// TIA Portal V17 export
// export: Created 2024-08-20T13:26:05.2375975Z, ExportSetting WithDefaults, DisplayName Totally Integrated Automation Portal, DisplayVersion V17 Update 4, DisplayName TIA Portal Openness, DisplayVersion V17 Update 4, DisplayName TIA Portal Version Control Interface, DisplayVersion V17, DisplayName STEP 7 Professional, DisplayVersion V17 Update 4, DisplayName STEP 7 Safety, DisplayVersion V17, DisplayName WinCC Advanced, DisplayVersion V17 Update 4
FUNCTION_BLOCK "DANFOSS_REV"   // FB206, LAD
TITLE = CONTROLE INVERSOR SINAMICS
{ S7_Optimized_Access := 'FALSE' }
VERSION : 0.1
// stored: AutoNumber false, IsIECCheckEnabled false, SetENOAutomatically false, UDAEnableTagReadback false
   VAR_INPUT
      DBNO : Int;   // Número do DB
      DBPOS : Int;   // Posição do DB
      MF1 : Bool;   // Motor em falha
      MF2 : Bool;   // Motor em falha
      HM : Bool;   // Habilita manual
      HA : Bool;   // Habilita automático
      HAR : Bool;   // Habilita automático reverso
      CMA : Bool;   // Comando liga automático
      CLM : Bool;   // Comando liga manual
      CLMR : Bool;   // Comando liga manual reverso
      CDM : Bool;   // Comando desliga manual
      CRF : Bool;   // Comando reset de falha
      CRTO : Bool;   // Comando reset tepo de operação
      CHC : Bool;   // Comando habilita controle de velocidade
      CHB : Bool;   // Comando habilita bloqueio
      CL1S : Bool;   // Pulso a cada 1 segundo
      SRC : Bool;   // Status rede de comunicação
      FMM : Real;   // Fundo de escala frequência do motor
      SPM : Real;   // Setpoint manual de velocidade
      SPA : Real;   // Setpoint automático de velocidade
   END_VAR
   VAR_OUTPUT
      YFL : Bool;   // Indicação de falha no inversor
      YFPP : Bool;   // Indicação de falha no acionamento
      YR : Bool;   // Indicação de chave na posição remota
      YSH : Bool;   // Indicação de motor ligado
      YF : Bool;   // Indicação de motor em falha
      CL : Bool;   // Comando liga motor
      REV : Bool;   // Indicação de motor ligado no sentido reverso
      CMD_RESET : Bool;   // Reset de falha
      IN18 : Bool;   // ENTRADA DIGITAL
      IN19 : Bool;   // ENTRADA DIGITAL
      IN27 : Bool;   // ENTRADA DIGITAL
      IN29 : Bool;   // ENTRADA DIGITAL
      IN32 : Bool;   // ENTRADA DIGITAL
      IN33 : Bool;   // ENTRADA DIGITAL
      IT : Real;   // Indicação de corrente
      ST : Real;   // Indicação de frequência
   END_VAR
   VAR_IN_OUT
      SEG : Int;   // Segundos de operação
      MIN : Int;   // Minutos de operação
      HOR : Int;   // Horas de operação
   END_VAR
   VAR DB_SPECIFIC
      STW { ExternalAccessible := 'False'; ExternalVisible := 'False'; ExternalWritable := 'False'} : Struct   // PALAVRA DE STATUS DO INVERSOR
         SpeddRef { ExternalAccessible := 'False'; ExternalVisible := 'False'; ExternalWritable := 'False'} : Bool;   // Velocidade=Setpoint
         BUS { ExternalAccessible := 'False'; ExternalVisible := 'False'; ExternalWritable := 'False'} : Bool;   // Controle pelo BUS
         FreqOK { ExternalAccessible := 'False'; ExternalVisible := 'False'; ExternalWritable := 'False'} : Bool;   // Frequecia OK
         Operation { ExternalAccessible := 'False'; ExternalVisible := 'False'; ExternalWritable := 'False'} : Bool;   // Em operação
         Drive { ExternalAccessible := 'False'; ExternalVisible := 'False'; ExternalWritable := 'False'} : Bool;   // Drive OK
         Voltage { ExternalAccessible := 'False'; ExternalVisible := 'False'; ExternalWritable := 'False'} : Bool;   // Tensão excedida
         Torque { ExternalAccessible := 'False'; ExternalVisible := 'False'; ExternalWritable := 'False'} : Bool;   // Torque excedido
         Thermal { ExternalAccessible := 'False'; ExternalVisible := 'False'; ExternalWritable := 'False'} : Bool;   // Térmico excedido
         Ready_forswitch_on { ExternalAccessible := 'False'; ExternalVisible := 'False'; ExternalWritable := 'False'} : Bool;   // Controle habilitado
         Ready { ExternalAccessible := 'False'; ExternalVisible := 'False'; ExternalWritable := 'False'} : Bool;   // Inversor pronto
         Running { ExternalAccessible := 'False'; ExternalVisible := 'False'; ExternalWritable := 'False'} : Bool;   // Em funcionamento
         Fault { ExternalAccessible := 'False'; ExternalVisible := 'False'; ExternalWritable := 'False'} : Bool;   // Falha ativa
         Error { ExternalAccessible := 'False'; ExternalVisible := 'False'; ExternalWritable := 'False'} : Bool;   // Erro ativo
         Reservado { ExternalAccessible := 'False'; ExternalVisible := 'False'; ExternalWritable := 'False'} : Bool;   // Reservado
         TripLock { ExternalAccessible := 'False'; ExternalVisible := 'False'; ExternalWritable := 'False'} : Bool;   // Inibição ativa
         Warning { ExternalAccessible := 'False'; ExternalVisible := 'False'; ExternalWritable := 'False'} : Bool;   // Advertência
      END_STRUCT;
      LPZD2 : Int;   // Velocidade do motor
      LPZD3 : Int;   // Corrente do motor
      LPZD4 : Struct   // Entradas digitais
         INX2 : Bool;   // Reservado
         INX3 : Bool;   // Reservado
         INX4 : Bool;   // Reservado
         INX5 : Bool;   // Reservado
         INX6 : Bool;   // Reservado
         INX7 : Bool;   // Reservado
         INX8 : Bool;   // Reservado
         INX9 : Bool;   // Reservado
         IN33 : Bool;   // Entrada terminal 33
         IN32 : Bool;   // Entrada terminal 32
         IN29 : Bool;   // Entrada terminal 29
         IN27 : Bool;   // Entrada terminal 27
         IN19 : Bool;   // Entrada terminal 19
         IN18 : Bool;   // Entrada terminal 18
         INX0 : Bool;   // Reservado
         INX1 : Bool;   // Reservado
      END_STRUCT;
      CTW { ExternalAccessible := 'False'; ExternalVisible := 'False'; ExternalWritable := 'False'} : Struct   // PALAVRA DE CONTROLE DO INVERSOR
         Jog { ExternalAccessible := 'False'; ExternalVisible := 'False'; ExternalWritable := 'False'} : Bool;   // Habilita jog
         RampSEL { ExternalAccessible := 'False'; ExternalVisible := 'False'; ExternalWritable := 'False'} : Bool;   // Seleção RAMPA1/2
         Control_plc { ExternalAccessible := 'False'; ExternalVisible := 'False'; ExternalWritable := 'False'} : Bool;   // Valida dados do PLC
         Relay1 { ExternalAccessible := 'False'; ExternalVisible := 'False'; ExternalWritable := 'False'} : Bool;   // Habilita partida sentido reverso
         Relay4 { ExternalAccessible := 'False'; ExternalVisible := 'False'; ExternalWritable := 'False'} : Bool;   // Controlador de velocidade habilitado
         Setup0 { ExternalAccessible := 'False'; ExternalVisible := 'False'; ExternalWritable := 'False'} : Bool;   // Seleção de setup bit0
         Setup1 { ExternalAccessible := 'False'; ExternalVisible := 'False'; ExternalWritable := 'False'} : Bool;   // Seleção de setup bit1
         Start_reverse { ExternalAccessible := 'False'; ExternalVisible := 'False'; ExternalWritable := 'False'} : Bool;   // Habilita partida sentido reverso
         LSB { ExternalAccessible := 'False'; ExternalVisible := 'False'; ExternalWritable := 'False'} : Bool;   // Seleção externa LSB
         MSB { ExternalAccessible := 'False'; ExternalVisible := 'False'; ExternalWritable := 'False'} : Bool;   // Seleção externa MSB
         DCbrakeRamp { ExternalAccessible := 'False'; ExternalVisible := 'False'; ExternalWritable := 'False'} : Bool;   // Freio DC/Rampa
         Coasting { ExternalAccessible := 'False'; ExternalVisible := 'False'; ExternalWritable := 'False'} : Bool;   // Liga motor
         Enable_Ramp { ExternalAccessible := 'False'; ExternalVisible := 'False'; ExternalWritable := 'False'} : Bool;   // Habilita rampa
         Enable_ramp_generator { ExternalAccessible := 'False'; ExternalVisible := 'False'; ExternalWritable := 'False'} : Bool;   // Habilita gerador de rampa
         Start { ExternalAccessible := 'False'; ExternalVisible := 'False'; ExternalWritable := 'False'} : Bool;   // Liga motor
         Reset { ExternalAccessible := 'False'; ExternalVisible := 'False'; ExternalWritable := 'False'} : Bool;   // Reconhecimento de falha
      END_STRUCT;
      CT_MotorReference : Int;   // Referência de velocidade
      EPZD3 : Int;   // Reserva
      EPZD4 : Int;   // Reserva
      RESET : Bool;   // Reset de falha
      AUX01 : Bool;   // Auxiliar utilizado na lógica
      AUX02 : Bool;   // Auxiliar utilizado na lógica
      AUX03 : Bool;   // Auxiliar utilizado na lógica
      AUX04 : Bool;   // Auxiliar utilizado na lógica
      AUX05 : Bool;   // Auxiliar utilizado na lógica
      AUX06 : Bool;   // Auxiliar utilizado na lógica
      AUX07 : Bool;   // Auxiliar utilizado na lógica
      AUX08 : Bool;   // Auxiliar utilizado na lógica
      AUX09 : Bool;   // Auxiliar utilizado na lógica
      AUX10 : Bool;   // Auxiliar utilizado na lógica
      P60S : Bool;   // Pulso de 60 segundos
      P60M : Bool;   // Pulso de 60 minutos
      PFHO : Bool;   // Pulso de limite de horas
      SPS : Real;   // Frequência para controle
      TPP1 { S7_SetPoint := 'True'} : TON_TIME;   // Temporizador falha no acionamento
      TPP2 { S7_SetPoint := 'True'} : TON_TIME;   // Temporizador falha no acionamento
      TR { S7_SetPoint := 'True'} : TON_TIME;   // Temporizador reset de falha
   END_VAR
   VAR_TEMP
      LIGADO : Bool;   // Ligado
      FALHA : Bool;   // Falha
      TEMP0 : Bool;
      TEMP1 : Bool;
      ET_TPP1 : Time;   // Efetivo temporizador
      ET_TPP2 : Time;   // Efetivo temporizador
      ET_TR : Time;   // Efetivo temporizador
      AUXDB : Int;   // Auxiliar movimentação do DB
      ST1 : Real;   // Frequência convertida
   END_VAR
   VAR_TEMP   // added for the SCL form of the ladder/FBD networks
      _w1 : Bool;
      _w2 : Bool;
      _w3 : Bool;
      _w4 : Bool;
   END_VAR
BEGIN

NETWORK
TITLE = Leitura de dados da rede
//CARREGA O ENDEREÇO DA PRIMEIRA WORD DE ENTRADA

      L     #DBNO;  // Carrega n° da DB
      T     #AUXDB;

      OPN   DB [#AUXDB];  // Abre DB

      L     #DBPOS;  // Multiplica valor da posição para acertar ponteiro (valor x 8bit´s)
      L     8;
      *I;
      LAR1;  // Carrega valor de ponteiro no registrador 1

      L     DBW [AR1, P#0.0];
      T     %DIW34;
      L     DBW [AR1, P#2.0];
      T     #LPZD2;
      L     DBW [AR1, P#4.0];
      T     #LPZD3;
      L     DBW [AR1, P#6.0];
      T     %DIW40;

NETWORK
TITLE = CONVERSÃO DA LEITURA DE FREQUÊNCIA/CORRENTE
      L     #LPZD2;
      ITD;
      DTR;
      L     #FMM;
      *R;
      L     16384.0;
      /R;
      T     #ST;

      L     #LPZD3;
      ITD;
      DTR;
      L     100.0;
      /R;
      T     #IT;

NETWORK
TITLE = STATUS DO INVERSOR
// VERIFICA ESTADO DO PRIMEIRO BYTE DA PALAVRA DE ENTRADA  (PZD)

      A     #STW.Fault;
      =     #YFL;  //ALARME DE FALHA NO INVERSOR

// LEITURA DAS ENTRADAS DIGITAIS

      A     #LPZD4.IN33;  // ENTRADA DIGITAL DE REMOTO
      A     #STW.BUS;
      =     #YR;
      =     #IN33;

      A     #LPZD4.IN18;  // TERMINAL 18
      =     #IN18;

      A     #LPZD4.IN19;  // TERMINAL 19
      =     #IN19;

      A     #LPZD4.IN27;  // TERMINAL 27
      =     #IN27;

      A     #LPZD4.IN32;  // TERMINAL 32
      =     #IN32;

      A     #LPZD4.IN29;  // TERMINAL 29
      =     #IN29;

REGION Network 4: STATUS DE LIGADO
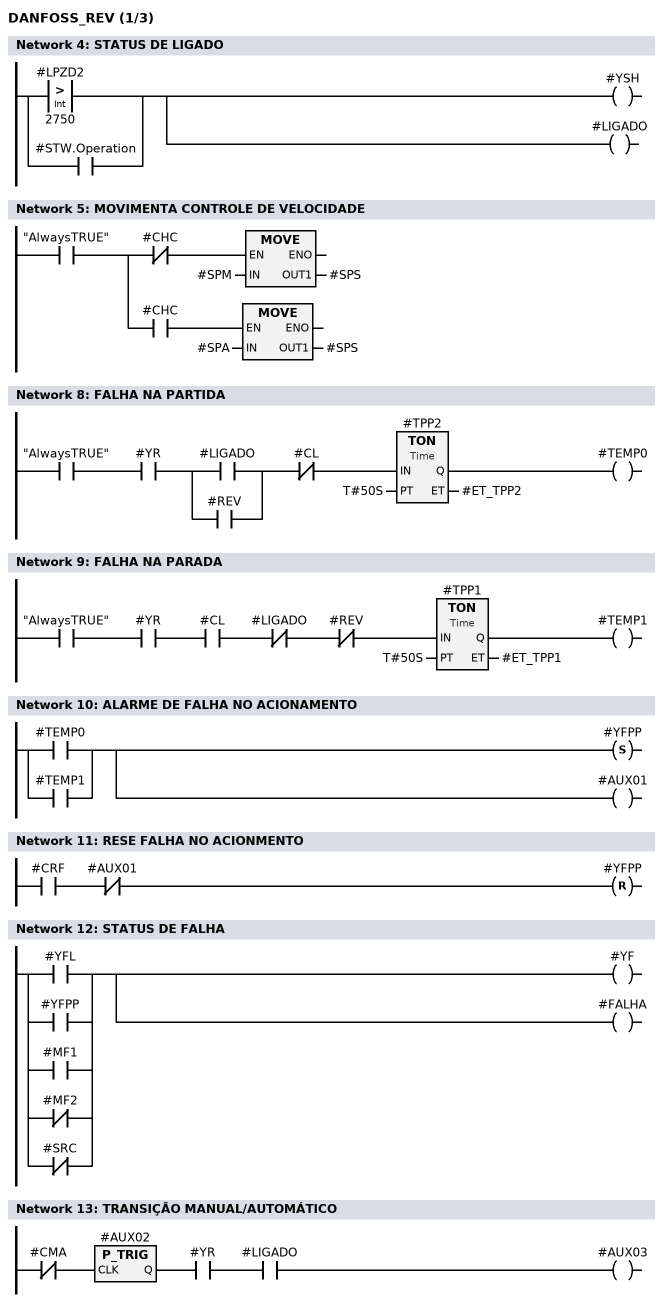
   RUNG wire#powerrail
      { S7_Templates := "SrcType := Int" } GT_Contact(in1 := #LPZD2, in2 := 2750)
      wire#w1
      Coil( #YSH )
   END_RUNG
   RUNG wire#powerrail
      Contact( #STW.Operation )
   END_RUNG wire#w1
   RUNG wire#w1
      Coil( #LIGADO )
   END_RUNG
   // the same network as SCL:
   #YSH := (#LPZD2 > 2750) OR #STW.Operation;
   #LIGADO := #YSH;
END_REGION

REGION Network 5: MOVIMENTA CONTROLE DE VELOCIDADE
   RUNG wire#powerrail
      Contact( "AlwaysTRUE" )
      wire#w1
      I_Contact( #CHC )
      { S7_GenerateENO := "TRUE" } Move(in := #SPM, out1 => #SPS)
   END_RUNG
   RUNG wire#w1
      Contact( #CHC )
      { S7_GenerateENO := "TRUE" } Move(in := #SPA, out1 => #SPS)
   END_RUNG
   // the same network as SCL:
   IF "AlwaysTRUE" AND NOT #CHC THEN #SPS := #SPM; END_IF;
   IF "AlwaysTRUE" AND #CHC THEN #SPS := #SPA; END_IF;
END_REGION

NETWORK
TITLE = Escreve setpoint de velocidade no inversor
      L     16384.0;  //Divide para encontrar a relação de conversão
      L     #SPS;
      *R;

      L     #FMM;  //Multiplica setpoint por fator para envio ao inversor
      /R;
      RND;
      T     #CT_MotorReference;


NETWORK
TITLE = ESCRITA DE DADOS NO INVERSOR
      +AR1  P#20.0;  //Carrega posição de escrita da DB

      L     %DIW42;
      T     DBW [AR1, P#0.0];  //Offset inicial
      L     #CT_MotorReference;
      T     DBW [AR1, P#2.0];


REGION Network 8: FALHA NA PARTIDA
   RUNG wire#powerrail
      Contact( "AlwaysTRUE" )
      Contact( #YR )
      wire#w1
      Contact( #LIGADO )
      wire#w2
      I_Contact( #CL )
      { S7_Templates := "time_type := Time" } #TPP2.TON(pt := T#50S, et => #ET_TPP2)
      Coil( #TEMP0 )
   END_RUNG
   RUNG wire#w1
      Contact( #REV )
   END_RUNG wire#w2
   // the same network as SCL:
   #TPP2(IN := "AlwaysTRUE" AND #YR AND (#LIGADO OR #REV) AND NOT #CL, PT := T#50S, ET => #ET_TPP2);   // TON
   #TEMP0 := #TPP2.Q;
END_REGION

REGION Network 9: FALHA NA PARADA
   RUNG wire#powerrail
      Contact( "AlwaysTRUE" )
      Contact( #YR )
      Contact( #CL )
      I_Contact( #LIGADO )
      I_Contact( #REV )
      { S7_Templates := "time_type := Time" } #TPP1.TON(pt := T#50S, et => #ET_TPP1)
      Coil( #TEMP1 )
   END_RUNG
   // the same network as SCL:
   #TPP1(IN := "AlwaysTRUE" AND #YR AND #CL AND NOT #LIGADO AND NOT #REV, PT := T#50S, ET => #ET_TPP1);   // TON
   #TEMP1 := #TPP1.Q;
END_REGION

REGION Network 10: ALARME DE FALHA NO ACIONAMENTO
   RUNG wire#powerrail
      Contact( #TEMP0 )
      wire#w1
      S_Coil( #YFPP )
   END_RUNG
   RUNG wire#powerrail
      Contact( #TEMP1 )
   END_RUNG wire#w1
   RUNG wire#w1
      Coil( #AUX01 )
   END_RUNG
   // the same network as SCL:
   #_w1 := #TEMP0 OR #TEMP1;
   IF #_w1 THEN #YFPP := TRUE; END_IF;
   #AUX01 := #_w1;
END_REGION

REGION Network 11: RESE FALHA NO ACIONMENTO
   RUNG wire#powerrail
      Contact( #CRF )
      I_Contact( #AUX01 )
      R_Coil( #YFPP )
   END_RUNG
   // the same network as SCL:
   IF #CRF AND NOT #AUX01 THEN #YFPP := FALSE; END_IF;
END_REGION

REGION Network 12: STATUS DE FALHA
   RUNG wire#powerrail
      Contact( #YFL )
      wire#w1
      Coil( #YF )
   END_RUNG
   RUNG wire#powerrail
      Contact( #YFPP )
   END_RUNG wire#w1
   RUNG wire#powerrail
      Contact( #MF1 )
   END_RUNG wire#w1
   RUNG wire#powerrail
      I_Contact( #MF2 )
   END_RUNG wire#w1
   RUNG wire#powerrail
      I_Contact( #SRC )
   END_RUNG wire#w1
   RUNG wire#w1
      Coil( #FALHA )
   END_RUNG
   // the same network as SCL:
   #YF := #YFL OR #YFPP OR #MF1 OR NOT #MF2 OR NOT #SRC;
   #FALHA := #YF;
END_REGION

REGION Network 13: TRANSIÇÃO MANUAL/AUTOMÁTICO
   RUNG wire#powerrail
      I_Contact( #CMA )
      P_Trig( #AUX02 )
      Contact( #YR )
      Contact( #LIGADO )
      Coil( #AUX03 )
   END_RUNG
   // the same network as SCL:
   #_w1 := NOT #CMA AND NOT #AUX02;   // rising edge
   #AUX02 := NOT #CMA;
   #AUX03 := #_w1 AND #YR AND #LIGADO;
END_REGION

REGION Network 14: COMANDO LIGA MANUAL SENTIDO DIRETO
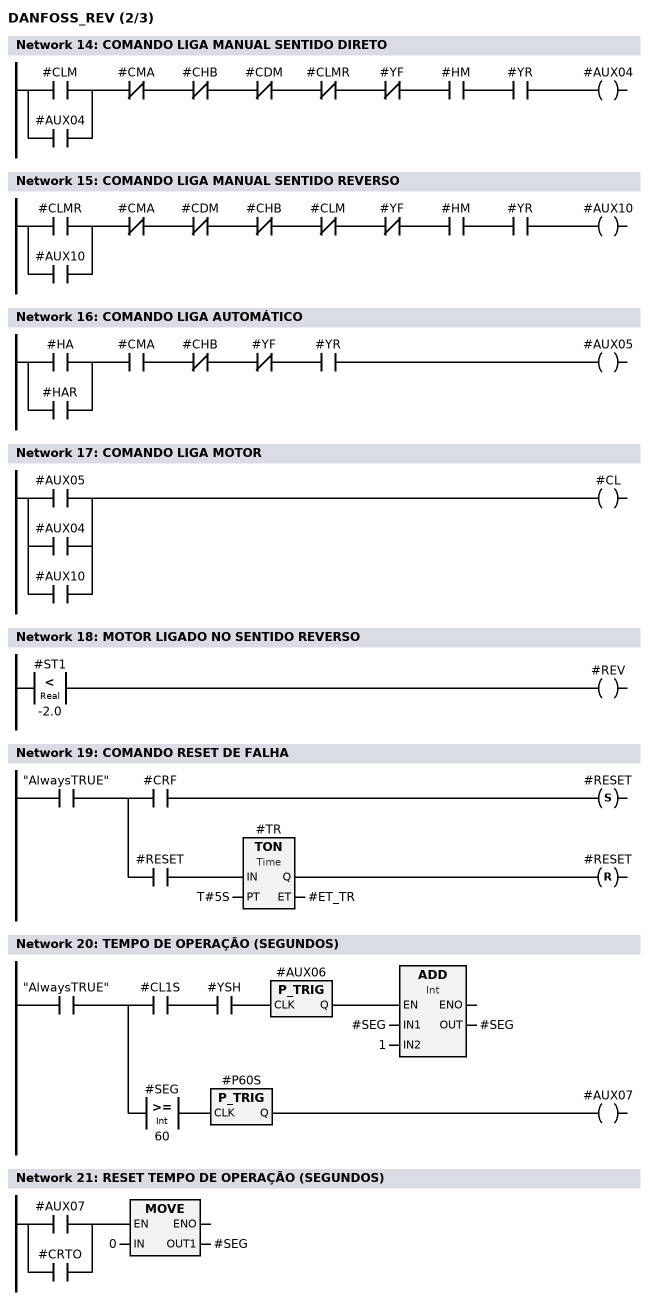
   RUNG wire#powerrail
      Contact( #CLM )
      wire#w1
      I_Contact( #CMA )
      I_Contact( #CHB )
      I_Contact( #CDM )
      I_Contact( #CLMR )
      I_Contact( #YF )
      Contact( #HM )
      Contact( #YR )
      Coil( #AUX04 )
   END_RUNG
   RUNG wire#powerrail
      Contact( #AUX04 )
   END_RUNG wire#w1
   // the same network as SCL:
   #AUX04 := (#CLM OR #AUX04) AND NOT #CMA AND NOT #CHB AND NOT #CDM AND NOT #CLMR AND NOT #YF AND #HM AND #YR;
END_REGION

REGION Network 15: COMANDO LIGA MANUAL SENTIDO REVERSO
   RUNG wire#powerrail
      Contact( #CLMR )
      wire#w1
      I_Contact( #CMA )
      I_Contact( #CDM )
      I_Contact( #CHB )
      I_Contact( #CLM )
      I_Contact( #YF )
      Contact( #HM )
      Contact( #YR )
      Coil( #AUX10 )
   END_RUNG
   RUNG wire#powerrail
      Contact( #AUX10 )
   END_RUNG wire#w1
   // the same network as SCL:
   #AUX10 := (#CLMR OR #AUX10) AND NOT #CMA AND NOT #CDM AND NOT #CHB AND NOT #CLM AND NOT #YF AND #HM AND #YR;
END_REGION

REGION Network 16: COMANDO LIGA AUTOMÁTICO
   RUNG wire#powerrail
      Contact( #HA )
      wire#w1
      Contact( #CMA )
      I_Contact( #CHB )
      I_Contact( #YF )
      Contact( #YR )
      Coil( #AUX05 )
   END_RUNG
   RUNG wire#powerrail
      Contact( #HAR )
   END_RUNG wire#w1
   // the same network as SCL:
   #AUX05 := (#HA OR #HAR) AND #CMA AND NOT #CHB AND NOT #YF AND #YR;
END_REGION

REGION Network 17: COMANDO LIGA MOTOR
   RUNG wire#powerrail
      Contact( #AUX05 )
      wire#w1
      Coil( #CL )
   END_RUNG
   RUNG wire#powerrail
      Contact( #AUX04 )
   END_RUNG wire#w1
   RUNG wire#powerrail
      Contact( #AUX10 )
   END_RUNG wire#w1
   // the same network as SCL:
   #CL := #AUX05 OR #AUX04 OR #AUX10;
END_REGION

REGION Network 18: MOTOR LIGADO NO SENTIDO REVERSO
   RUNG wire#powerrail
      { S7_Templates := "SrcType := Real" } LT_Contact(in1 := #ST1, in2 := -2.0)
      Coil( #REV )
   END_RUNG
   // the same network as SCL:
   #REV := #ST1 < (-2.0);
END_REGION

REGION Network 19: COMANDO RESET DE FALHA
   RUNG wire#powerrail
      Contact( "AlwaysTRUE" )
      wire#w1
      Contact( #CRF )
      S_Coil( #RESET )
   END_RUNG
   RUNG wire#w1
      Contact( #RESET )
      { S7_Templates := "time_type := Time" } #TR.TON(pt := T#5S, et => #ET_TR)
      R_Coil( #RESET )
   END_RUNG
   // the same network as SCL:
   IF "AlwaysTRUE" AND #CRF THEN #RESET := TRUE; END_IF;
   #TR(IN := "AlwaysTRUE" AND #RESET, PT := T#5S, ET => #ET_TR);   // TON
   IF #TR.Q THEN #RESET := FALSE; END_IF;
END_REGION

REGION Network 20: TEMPO DE OPERAÇÃO (SEGUNDOS)
   RUNG wire#powerrail
      Contact( "AlwaysTRUE" )
      wire#w1
      Contact( #CL1S )
      Contact( #YSH )
      P_Trig( #AUX06 )
      { S7_Templates := "SrcType := Int"; S7_GenerateENO := "TRUE" } Add(in1 := #SEG, in2 := 1, out => #SEG)
   END_RUNG
   RUNG wire#w1
      { S7_Templates := "SrcType := Int" } GE_Contact(in1 := #SEG, in2 := 60)
      P_Trig( #P60S )
      Coil( #AUX07 )
   END_RUNG
   // the same network as SCL:
   #_w1 := "AlwaysTRUE" AND #CL1S AND #YSH;
   #_w2 := #_w1 AND NOT #AUX06;   // rising edge
   #AUX06 := #_w1;
   IF #_w2 THEN #SEG := #SEG + 1; END_IF;
   #_w3 := "AlwaysTRUE" AND (#SEG >= 60);
   #_w4 := #_w3 AND NOT #P60S;   // rising edge
   #P60S := #_w3;
   #AUX07 := #_w4;
END_REGION

REGION Network 21: RESET TEMPO DE OPERAÇÃO (SEGUNDOS)
   RUNG wire#powerrail
      Contact( #AUX07 )
      wire#w1
      { S7_GenerateENO := "TRUE" } Move(in := 0, out1 => #SEG)
   END_RUNG
   RUNG wire#powerrail
      Contact( #CRTO )
   END_RUNG wire#w1
   // the same network as SCL:
   IF #AUX07 OR #CRTO THEN #SEG := 0; END_IF;
END_REGION

REGION Network 22: TEMPO DE OPERAÇÃO (MINUTOS)
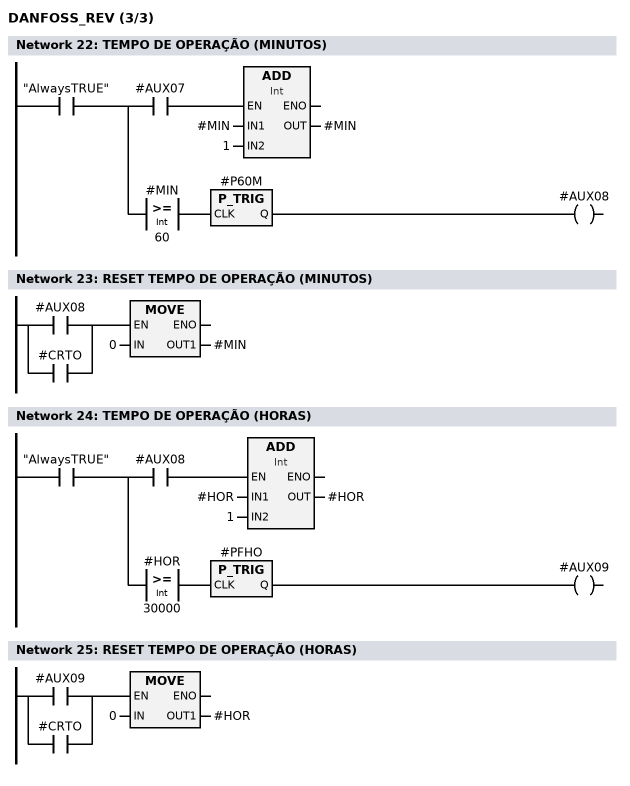
   RUNG wire#powerrail
      Contact( "AlwaysTRUE" )
      wire#w1
      Contact( #AUX07 )
      { S7_Templates := "SrcType := Int"; S7_GenerateENO := "TRUE" } Add(in1 := #MIN, in2 := 1, out => #MIN)
   END_RUNG
   RUNG wire#w1
      { S7_Templates := "SrcType := Int" } GE_Contact(in1 := #MIN, in2 := 60)
      P_Trig( #P60M )
      Coil( #AUX08 )
   END_RUNG
   // the same network as SCL:
   IF "AlwaysTRUE" AND #AUX07 THEN #MIN := #MIN + 1; END_IF;
   #_w1 := "AlwaysTRUE" AND (#MIN >= 60);
   #_w2 := #_w1 AND NOT #P60M;   // rising edge
   #P60M := #_w1;
   #AUX08 := #_w2;
END_REGION

REGION Network 23: RESET TEMPO DE OPERAÇÃO (MINUTOS)
   RUNG wire#powerrail
      Contact( #AUX08 )
      wire#w1
      { S7_GenerateENO := "TRUE" } Move(in := 0, out1 => #MIN)
   END_RUNG
   RUNG wire#powerrail
      Contact( #CRTO )
   END_RUNG wire#w1
   // the same network as SCL:
   IF #AUX08 OR #CRTO THEN #MIN := 0; END_IF;
END_REGION

REGION Network 24: TEMPO DE OPERAÇÃO (HORAS)
   RUNG wire#powerrail
      Contact( "AlwaysTRUE" )
      wire#w1
      Contact( #AUX08 )
      { S7_Templates := "SrcType := Int"; S7_GenerateENO := "TRUE" } Add(in1 := #HOR, in2 := 1, out => #HOR)
   END_RUNG
   RUNG wire#w1
      { S7_Templates := "SrcType := Int" } GE_Contact(in1 := #HOR, in2 := 30000)
      P_Trig( #PFHO )
      Coil( #AUX09 )
   END_RUNG
   // the same network as SCL:
   IF "AlwaysTRUE" AND #AUX08 THEN #HOR := #HOR + 1; END_IF;
   #_w1 := "AlwaysTRUE" AND (#HOR >= 30000);
   #_w2 := #_w1 AND NOT #PFHO;   // rising edge
   #PFHO := #_w1;
   #AUX09 := #_w2;
END_REGION

REGION Network 25: RESET TEMPO DE OPERAÇÃO (HORAS)
   RUNG wire#powerrail
      Contact( #AUX09 )
      wire#w1
      { S7_GenerateENO := "TRUE" } Move(in := 0, out1 => #HOR)
   END_RUNG
   RUNG wire#powerrail
      Contact( #CRTO )
   END_RUNG wire#w1
   // the same network as SCL:
   IF #AUX09 OR #CRTO THEN #HOR := 0; END_IF;
END_REGION

NETWORK
TITLE = ESCRITA DOS DADOS NO INVERSOR (PALAVRA DE COMANDO)
      A     "AlwaysTRUE";
      =     #CTW.DCbrakeRamp;
      =     #CTW.Coasting;
      =     #CTW.Enable_Ramp;
      =     #CTW.Enable_ramp_generator;
      =     #CTW.Control_plc;  //Valida setpoint


      A     #CL;
      =     #CTW.Start;  //LIGA/DESL

      A     #CL;
      A     #AUX10;
      A     #HAR;
      =     #CTW.Start_reverse;  //LIGA/DESL REVERSO


      A     #RESET;
      AN    #CL;
      =     #CTW.Reset;  //RESET
END_FUNCTION_BLOCK
